// TIA Portal V20 export
DATA_BLOCK "LPFE_InterfaceChannels"   // DB242
TITLE = Buffer of RequestOrderInfo messages
// Contains Interface channel components for ToHost and Txn channels
// stored: Access Published, MemoryReserve 100, Namespace PFE
   VAR
      toHostChannels { ExternalVisible := 'False'} : Array[0.._.LE_NUMBER_OF_INTERFACE_BUFFERS] of "LPFE_typeRequestChannel";   // Channels for request/response messages
      txnChannel { ExternalAccessible := 'False'; ExternalVisible := 'False'; ExternalWritable := 'False'; S7_SetPoint := 'True'} : "LPFE_typePFEDataOutChannel";   // Channels for outbound messages
   END_VAR
BEGIN
END_DATA_BLOCK
